// TIA Portal V18 export
DATA_BLOCK "!!nameOfDB2$$"   // DB33, F_DB
{ S7_Optimized_Access := 'TRUE' }
   VAR
      AlwaysFALSE : Bool;
      AlwaysTRUE : Bool := TRUE;
      "!!ITERATOR_STRINGS$$" : Bool;
   END_VAR
BEGIN
END_DATA_BLOCK
